Omron Sysmac Studio project Test_ZW5000 (Sysmac Studio 1.47.0.64008, StandardProject)

# Controller new_Controller_0: NX102-9020 version 1.31
Units and slaves: Unit 1 : NX-PF0730 (N1)
Task PrimaryTask (priority 4, period or condition 2000): Program0
Library OmronLib_DIM_Measurement_V1_1 1.1.0 (contents left out)
Library OmronLib_DIM_PointMeasurement_V1_1 1.1.0 (contents left out)
Library OmronLib_DIM_LineMeasurement_V2_0 2.0.0 (contents left out)

VAR_GLOBAL
    ZW001_STABILITY : BOOL;  (* at ECAT://node#1/Sensor Head Status Signal2/STABILITY *)
    ZW001_Output_Data_1 : DINT;  (* at ECAT://node#1/Output Data 1 *)
    ZW001_Real_Data : REAL;
    ZW001_Real_Data_mm : REAL;
END_VAR

PROGRAM Program0
VAR
    ZW001_Real_us : REAL;
END_VAR
VAR_EXTERNAL
    ZW001_STABILITY : BOOL;
    ZW001_Output_Data_1 : DINT;
    ZW001_Real_Data_mm : REAL;
END_VAR

(* Section Section0: ladder, written here as Structured Text *)

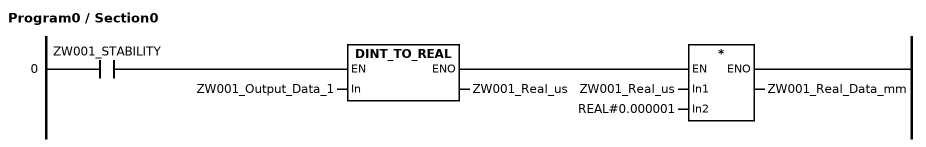
(* Rung 0 *)
IF ZW001_STABILITY THEN
    ZW001_Real_us := DINT_TO_REAL(In := ZW001_Output_Data_1);
    ZW001_Real_Data_mm := ZW001_Real_us * REAL#0.000001;
END_IF;
END_PROGRAM